{attribute 'qualified_only'}
{attribute 'strict'}
TYPE E_MoverTransitionState :
(

	MoveToPick  := 11,
	Picking     := 12,
	MoveToPlace := 13,
	Placing     := 14
);
END_TYPE

(* stored: Version 1.1.0.1, ProductVersion 3.1.4024.12
   DUT E_MoverTransitionState: Id {331c631a-7bd6-4a87-b502-e5c9c2d28555} *)
